END_VAR
VAR_INPUT
	bWlaczPrzyciski								: BOOL;
END_VAR
    Rectangle (0,0 901x401)
    Rectangle (10,10 881x241)
    Frame (210,20 114x44), invisible if: not GVL_StanMaszyny.fbStanMaszyny.arrVisuTryb[GVL_StanMaszyny.fbStanMaszyny.iNumerTrybuPracy][12]
        shows Visu_StanMaszyny_AktualyStan(bNacisniety := GVL_StanMaszyny.fbStanMaszyny.bUnholdingZakonczone, stVisuStan := GVL_StanMaszyny.fbStanMaszyny.arrVisuStany [12])
    Frame (400,20 114x44), invisible if: not GVL_StanMaszyny.fbStanMaszyny.arrVisuTryb[GVL_StanMaszyny.fbStanMaszyny.iNumerTrybuPracy][11]
        shows Visu_StanMaszyny_AktualyStan_BezNaciskania(stVisuStan := GVL_StanMaszyny.fbStanMaszyny.arrVisuStany [11])
    Frame (580,20 114x44), invisible if: not GVL_StanMaszyny.fbStanMaszyny.arrVisuTryb[GVL_StanMaszyny.fbStanMaszyny.iNumerTrybuPracy][10]
        shows Visu_StanMaszyny_AktualyStan(bNacisniety := GVL_StanMaszyny.fbStanMaszyny.bHoldingZakonczone, stVisuStan := GVL_StanMaszyny.fbStanMaszyny.arrVisuStany [10])
    Frame (20,110 114x44), invisible if: not GVL_StanMaszyny.fbStanMaszyny.arrVisuTryb[GVL_StanMaszyny.fbStanMaszyny.iNumerTrybuPracy][4]
        shows Visu_StanMaszyny_AktualyStan_BezNaciskania(stVisuStan := GVL_StanMaszyny.fbStanMaszyny.arrVisuStany [4])
    Frame (210,110 114x44), invisible if: not GVL_StanMaszyny.fbStanMaszyny.arrVisuTryb[GVL_StanMaszyny.fbStanMaszyny.iNumerTrybuPracy][3]
        shows Visu_StanMaszyny_AktualyStan(bNacisniety := GVL_StanMaszyny.fbStanMaszyny.bStartingZakonczone, stVisuStan := GVL_StanMaszyny.fbStanMaszyny.arrVisuStany [3])
    Frame (400,110 114x44), invisible if: not GVL_StanMaszyny.fbStanMaszyny.arrVisuTryb[GVL_StanMaszyny.fbStanMaszyny.iNumerTrybuPracy][6]
        shows Visu_StanMaszyny_AktualyStan_BezNaciskania(stVisuStan := GVL_StanMaszyny.fbStanMaszyny.arrVisuStany [6])
    Frame (580,110 114x44), invisible if: not GVL_StanMaszyny.fbStanMaszyny.arrVisuTryb[GVL_StanMaszyny.fbStanMaszyny.iNumerTrybuPracy][16]
        shows Visu_StanMaszyny_AktualyStan(bNacisniety := GVL_StanMaszyny.fbStanMaszyny.bCompletingZakonczone, stVisuStan := GVL_StanMaszyny.fbStanMaszyny.arrVisuStany [16])
    Frame (765,110 114x44), invisible if: not GVL_StanMaszyny.fbStanMaszyny.arrVisuTryb[GVL_StanMaszyny.fbStanMaszyny.iNumerTrybuPracy][17]
        shows Visu_StanMaszyny_AktualyStan_BezNaciskania(stVisuStan := GVL_StanMaszyny.fbStanMaszyny.arrVisuStany [17])
    Frame (20,200 114x44), invisible if: not GVL_StanMaszyny.fbStanMaszyny.arrVisuTryb[GVL_StanMaszyny.fbStanMaszyny.iNumerTrybuPracy][15]
        shows Visu_StanMaszyny_AktualyStan(bNacisniety := GVL_StanMaszyny.fbStanMaszyny.bResetingSkonczone, stVisuStan := GVL_StanMaszyny.fbStanMaszyny.arrVisuStany [15])
    Frame (210,200 114x44), invisible if: not GVL_StanMaszyny.fbStanMaszyny.arrVisuTryb[GVL_StanMaszyny.fbStanMaszyny.iNumerTrybuPracy][14]
        shows Visu_StanMaszyny_AktualyStan(bNacisniety := GVL_StanMaszyny.fbStanMaszyny.bUnsuspendingZakonczone, stVisuStan := GVL_StanMaszyny.fbStanMaszyny.arrVisuStany [14])
    Frame (400,200 114x44), invisible if: not GVL_StanMaszyny.fbStanMaszyny.arrVisuTryb[GVL_StanMaszyny.fbStanMaszyny.iNumerTrybuPracy][5]
        shows Visu_StanMaszyny_AktualyStan_BezNaciskania(stVisuStan := GVL_StanMaszyny.fbStanMaszyny.arrVisuStany [5])
    Frame (580,200 114x44), invisible if: not GVL_StanMaszyny.fbStanMaszyny.arrVisuTryb[GVL_StanMaszyny.fbStanMaszyny.iNumerTrybuPracy][13]
        shows Visu_StanMaszyny_AktualyStan(bNacisniety := GVL_StanMaszyny.fbStanMaszyny.bSuspendingZakonczone, stVisuStan := GVL_StanMaszyny.fbStanMaszyny.arrVisuStany [13])
    Frame (20,340 114x44), invisible if: not GVL_StanMaszyny.fbStanMaszyny.arrVisuTryb[GVL_StanMaszyny.fbStanMaszyny.iNumerTrybuPracy][2]
        shows Visu_StanMaszyny_AktualyStan_BezNaciskania(stVisuStan := GVL_StanMaszyny.fbStanMaszyny.arrVisuStany [2])
    Frame (210,340 114x44), invisible if: not GVL_StanMaszyny.fbStanMaszyny.arrVisuTryb[GVL_StanMaszyny.fbStanMaszyny.iNumerTrybuPracy][7]
        shows Visu_StanMaszyny_AktualyStan(bNacisniety := GVL_StanMaszyny.fbStanMaszyny.bStoppingZakonczone, stVisuStan := GVL_StanMaszyny.fbStanMaszyny.arrVisuStany [7])
    Frame (400,340 114x44), invisible if: not GVL_StanMaszyny.fbStanMaszyny.arrVisuTryb[GVL_StanMaszyny.fbStanMaszyny.iNumerTrybuPracy][1]
        shows Visu_StanMaszyny_AktualyStan(bNacisniety := GVL_StanMaszyny.fbStanMaszyny.bClearingZakonczone, stVisuStan := GVL_StanMaszyny.fbStanMaszyny.arrVisuStany [1])
    Rectangle (550,320 351x81)
    Frame (580,340 114x44), invisible if: not GVL_StanMaszyny.fbStanMaszyny.arrVisuTryb[GVL_StanMaszyny.fbStanMaszyny.iNumerTrybuPracy][9]
        shows Visu_StanMaszyny_AktualyStan_BezNaciskania(stVisuStan := GVL_StanMaszyny.fbStanMaszyny.arrVisuStany [9])
    Frame (765,340 114x44), invisible if: not GVL_StanMaszyny.fbStanMaszyny.arrVisuTryb[GVL_StanMaszyny.fbStanMaszyny.iNumerTrybuPracy][8]
        shows Visu_StanMaszyny_AktualyStan(bNacisniety := GVL_StanMaszyny.fbStanMaszyny.bAbortingZakonczone, stVisuStan := GVL_StanMaszyny.fbStanMaszyny.arrVisuStany [8])
END_VISUALIZATION

// ---- POUs/90 - Stan Maszyny/Visu/Visu_StanMaszyny_DiagramZPrzyciskami.TcVIS
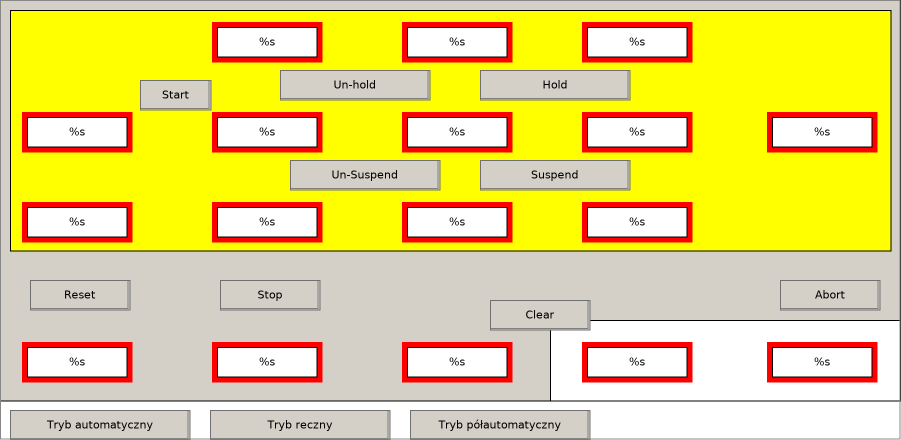
VISUALIZATION Visu_StanMaszyny_DiagramZPrzyciskami  // 901x440
VAR_IN_OUT
	
END_VAR
VAR_INPUT
	bWlaczPrzyciski								: BOOL;
END_VAR
    Frame (0,0 901x401)
        shows Visu_StanMaszyny_Diagram(bWlaczPrzyciski := bWlaczPrzyciski)
    Button (140,80 71x30), "Start", colour toggle: GVL_Elementy.fbPrzysciskStart.bPodswietlenie
        tap GVL_StanMaszyny.bStart
    Button (220,280 100x30), "Stop", colour toggle: GVL_Elementy.fbPrzyciskStop.bPodswietlenie
        tap GVL_StanMaszyny.bStop
    Button (30,280 100x30), "Reset"
        tap GVL_StanMaszyny.bReset
    Button (780,280 100x30), "Abort"
        tap GVL_StanMaszyny.bAbort
    Button (480,70 150x30), "Hold", invisible if: not GVL_StanMaszyny.fbStanMaszyny.arrVisuTryb[GVL_StanMaszyny.fbStanMaszyny.iNumerTrybuPracy][11]
        tap GVL_StanMaszyny.bHold
    Button (280,70 150x30), "Un-hold", invisible if: not GVL_StanMaszyny.fbStanMaszyny.arrVisuTryb[GVL_StanMaszyny.fbStanMaszyny.iNumerTrybuPracy][11]
        tap GVL_StanMaszyny.bUnhold
    Button (480,160 150x30), "Suspend", invisible if: not GVL_StanMaszyny.fbStanMaszyny.arrVisuTryb[GVL_StanMaszyny.fbStanMaszyny.iNumerTrybuPracy][5]
        tap GVL_StanMaszyny.bSuspend
    Button (290,160 150x30), "Un-Suspend", invisible if: not GVL_StanMaszyny.fbStanMaszyny.arrVisuTryb[GVL_StanMaszyny.fbStanMaszyny.iNumerTrybuPracy][5]
        tap GVL_StanMaszyny.bUnsuspend
    Button (10,410 180x30), "Tryb automatyczny", colour toggle: GVL_StanMaszyny.eTrybPracy = E_PMLUnitMode.AUTOMATIC, input disabled if: not (GVL_StanMaszyny.fbStanMaszyny.eStan = E_PMLState.ABORTED or GVL_StanMaszyny.fbStanMaszyny.eStan = E_PMLState.STOPPED)
        OnMouseDown: execute { GVL_StanMaszyny.eTrybPracy	:= E_PMLUnitMode.AUTOMATIC; }
    Button (210,410 180x30), "Tryb reczny", colour toggle: GVL_StanMaszyny.eTrybPracy = E_PMLUnitMode.MANUAL, input disabled if: not (GVL_StanMaszyny.fbStanMaszyny.eStan = E_PMLState.ABORTED or GVL_StanMaszyny.fbStanMaszyny.eStan = E_PMLState.STOPPED)
        OnMouseDown: execute { GVL_StanMaszyny.eTrybPracy	:= E_PMLUnitMode.MANUAL; }
    Button (490,300 100x30), "Clear"
        tap GVL_StanMaszyny.bClear
    Button (410,410 180x30), "Tryb półautomatyczny", colour toggle: GVL_StanMaszyny.eTrybPracy = E_PMLUnitMode.SEMIAUTOMATIC, input disabled if: not (GVL_StanMaszyny.fbStanMaszyny.eStan = E_PMLState.ABORTED or GVL_StanMaszyny.fbStanMaszyny.eStan = E_PMLState.STOPPED)
        OnMouseDown: execute { GVL_StanMaszyny.eTrybPracy	:= E_PMLUnitMode.SEMIAUTOMATIC; }
END_VISUALIZATION

// ---- POUs/95 - Logowanie bledow/Wizualizacja/Visu_LogowanieBledow_Tabela.TcVIS
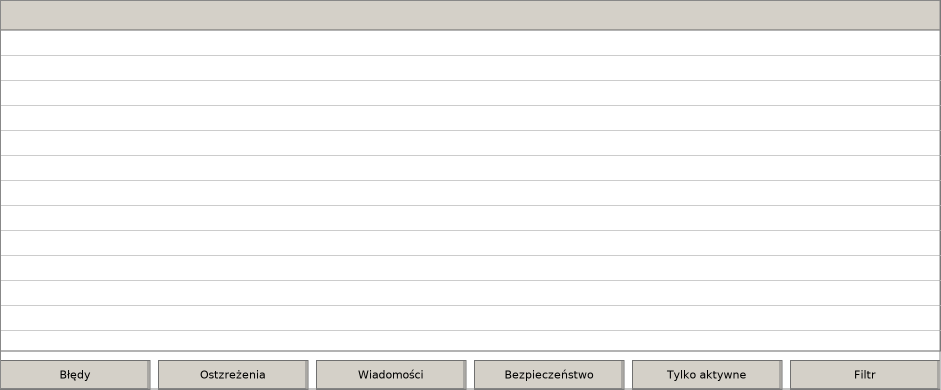
VISUALIZATION Visu_LogowanieBledow_Tabela  // 941x390
VAR_IN_OUT
	stParametry								: DUT_LogowanieBledow_WyswietlanieParametry;
END_VAR
    Table (0,0 941x351), data array: GVL_LogowanieBledow.fbLoger.arrTablicaWyswietlana
        p3854506369: GVL_LogowanieBledow.fbLoger.arrTablicaWyswietlana[INDEX].sNrKomponentu
        p1892666644: GVL_LogowanieBledow.fbLoger.arrTablicaWyswietlana[INDEX].sKodBledu
        p338671338: GVL_LogowanieBledow.fbLoger.arrTablicaWyswietlana[INDEX].byRodzajZdarzenia
        p2170511999: GVL_LogowanieBledow.fbLoger.arrTablicaWyswietlana[INDEX].sOpis
        p3723444502: GVL_LogowanieBledow.fbLoger.arrTablicaWyswietlana[INDEX].dtDataStart
        p1218418051: GVL_LogowanieBledow.fbLoger.arrTablicaWyswietlana[INDEX].dtDataKoniec
        p746581629: GVL_LogowanieBledow.fbLoger.arrTablicaWyswietlana[INDEX].dwKolor
        p2232123230: Nr Elem.
        p2237128397: Data start
        p505689113: Data koniec
        Columns.Column.[3].Template: 16#FF000000 OR (GVL_LogowanieBledow.fbLoger.arrTablicaWyswietlana[INDEX].dwKolor)
    Button (632,360 150x30), "Tylko aktywne", colour toggle: stParametry.bFiltrAktywne
        toggle stParametry.bFiltrAktywne
    Button (0,360 150x30), "Błędy", colour toggle: stParametry.bFiltrRodzaj and stParametry.byFiltrRodzaj = 1
        OnMouseDown: execute {
            (*
            IF (NOT stParametry.bFiltrRodzaj) THEN
            	stParametry.bFiltrRodzaj := TRUE;
            	stParametry.byFiltrRodzaj := 1;
            ELSE
            	stParametry.bFiltrRodzaj := FALSE;
            END_IF
            *)
        }
    Button (158,360 150x30), "Ostzreżenia", colour toggle: stParametry.bFiltrRodzaj and stParametry.byFiltrRodzaj = 2
        OnMouseDown: execute {
            (*
            IF (NOT stParametry.bFiltrRodzaj) THEN
            	stParametry.bFiltrRodzaj := TRUE;
            	stParametry.byFiltrRodzaj := 2;
            ELSE
            	stParametry.bFiltrRodzaj := FALSE;
            END_IF
            *)
        }
    Button (316,360 150x30), "Wiadomości", colour toggle: stParametry.bFiltrRodzaj and stParametry.byFiltrRodzaj = 3
        OnMouseDown: execute {
            (*
            IF (NOT stParametry.bFiltrRodzaj) THEN
            	stParametry.bFiltrRodzaj := TRUE;
            	stParametry.byFiltrRodzaj := 3;
            ELSE
            	stParametry.bFiltrRodzaj := FALSE;
            END_IF
            *)
        }
    Button (474,360 150x30), "Bezpieczeństwo", colour toggle: stParametry.bFiltrRodzaj and stParametry.byFiltrRodzaj = 4
        OnMouseDown: execute {
            (*
            IF (NOT stParametry.bFiltrRodzaj) THEN
            	stParametry.bFiltrRodzaj := TRUE;
            	stParametry.byFiltrRodzaj := 4;
            ELSE
            	stParametry.bFiltrRodzaj := FALSE;
            END_IF
            *)
        }
    Button (790,360 150x30), "Filtr"
END_VISUALIZATION

// ---- VISUs/OknoGlowne.TcVIS
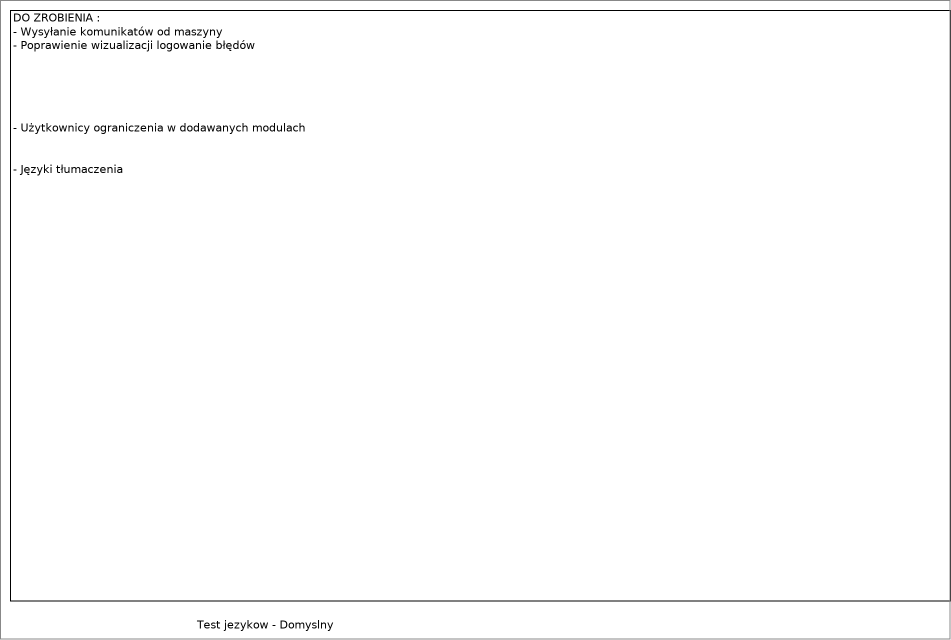
VISUALIZATION OknoGlowne  // 951x640
    Rectangle (10,10 941x591), "DO ZROBIENIA : - Wysyłanie komunikatów od maszyny - Poprawienie wizualizacji logowanie błędów - Użytkownicy ograniczenia w dodawanych modulach - Języki tłumaczenia"
    Label (50,610 431x30), "Test jezykow - Domyslny"
END_VISUALIZATION

// ---- VISUs/Symulacja.TcVIS
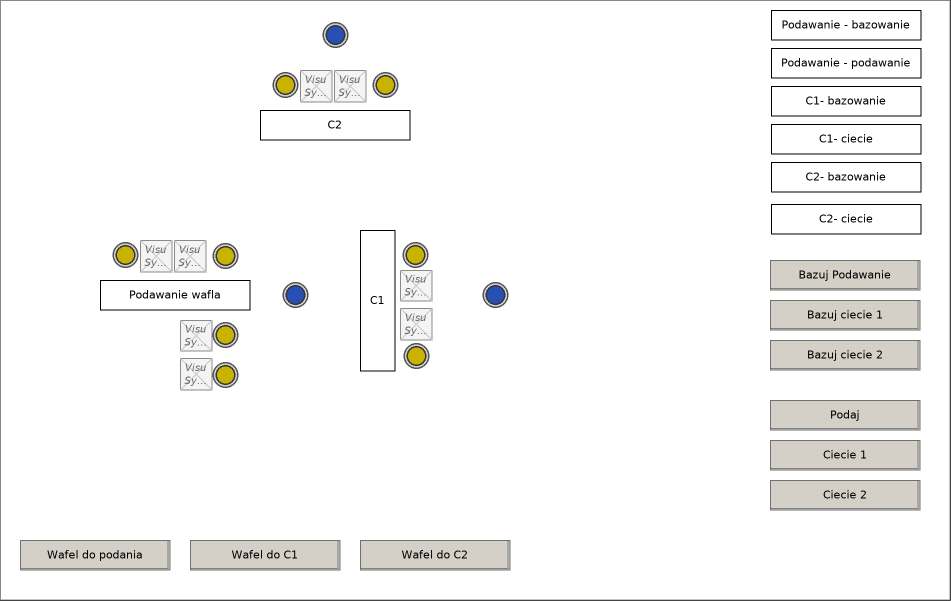
VISUALIZATION Symulacja  // 951x601
VAR_IN_OUT
	stDane									: DUT_Wizualizacja_SymulacjaDane;
END_VAR
    Line (950,0) (950,600)
    Line (0,600) (950,600)
    Rectangle (100,280 150x30), "Podawanie wafla"
    Rectangle (360,230 35x141), "C1"
    Rectangle (260,110 150x30), "C2"
    Lamp1 (401,341 31x30), variable: stDane.bCiecie1_Poczatek, style: Lamp-Lamp1-Yellow
    Lamp1 (400,240 31x30), variable: stDane.bCiecie1_Koniec, style: Lamp-Lamp1-Yellow
    Lamp1 (270,70 31x30), variable: stDane.bCiecie2_Poczatek, style: Lamp-Lamp1-Yellow
    Lamp1 (370,70 31x30), variable: stDane.bCiecie2_Koniec, style: Lamp-Lamp1-Yellow
    Lamp1 (110,240 31x30), variable: stDane.bPodawaniePrzesuwanieKoniec, style: Lamp-Lamp1-Yellow
    Lamp1 (210,241 31x30), variable: stDane.bPodawaniePrzesuwaniePoczatek, style: Lamp-Lamp1-Yellow
    Lamp1 (210,320 31x30), variable: stDane.bPodawanieZabierakKoniec, style: Lamp-Lamp1-Yellow
    Lamp1 (210,360 31x30), variable: stDane.bPodawanieZabierakPoczatek, style: Lamp-Lamp1-Yellow
    Lamp1 (280,280 31x30), variable: stDane.bCzujnikWaflaDoPodania, style: Lamp-Lamp1-Blue
    Lamp1 (480,280 31x30), variable: stDane.bCzujnikWaflaDoCiecia1, style: Lamp-Lamp1-Blue
    Lamp1 (320,20 31x30), variable: stDane.bCzujnikWaflaDoCiecia2, style: Lamp-Lamp1-Blue
    Rectangle (771,10 150x30), "Podawanie - bazowanie", colour toggle: stDane.stStanySilownikow.bPodawanie_Bazowanie
    Rectangle (771,48 150x30), "Podawanie - podawanie", colour toggle: stDane.stStanySilownikow.bPodawanie_Podawanie
    Rectangle (771,86 150x30), "C1- bazowanie", colour toggle: stDane.stStanySilownikow.bCiecie1_Bazowanie
    Rectangle (771,124 150x30), "C1- ciecie", colour toggle: stDane.stStanySilownikow.bCiecie1_Ciecie
    Rectangle (771,162 150x30), "C2- bazowanie", colour toggle: stDane.stStanySilownikow.bCiecie2_Bazowanie
    Rectangle (771,204 150x30), "C2- ciecie", colour toggle: stDane.stStanySilownikow.bCiecie2_Ciecie
    Image (180,358 32x32), invisible if: Not stDane.stStanySilownikow.bPodawanie_Zabierak_WStronePoczatku, image: VisuSymbols.Symbols.ArrowBoldDown
    Image (180,320 32x31), invisible if: Not stDane.stStanySilownikow.bPodawanie_zabierak_WStroneKonca, image: VisuSymbols.Symbols.ArrowBoldUp
    Image (140,240 32x32), invisible if: Not stDane.stStanySilownikow.bPodawanie_Przesuwanie_WStroneKonca, image: VisuSymbols.Symbols.ArrowBoldLeft
    Image (174,240 32x32), invisible if: Not stDane.stStanySilownikow.bPodawanie_Przesuwanie_WStronePoczatku, image: VisuSymbols.Symbols.ArrowBoldRight
    Image (400,308 32x32), invisible if: Not stDane.stStanySilownikow.bCiecie1_Naped_WStronePoczatku, image: VisuSymbols.Symbols.ArrowBoldDown
    Image (400,270 32x31), invisible if: Not stDane.stStanySilownikow.bCiecie1_Naped_WStroneKonca, image: VisuSymbols.Symbols.ArrowBoldUp
    Image (300,70 32x32), invisible if: Not stDane.stStanySilownikow.bCiecie2_Naped_WStronePoczatku, image: VisuSymbols.Symbols.ArrowBoldLeft
    Image (334,70 32x32), invisible if: Not stDane.stStanySilownikow.bCiecie2_Naped_WStroneKonca, image: VisuSymbols.Symbols.ArrowBoldRight
    Button (770,260 150x30), "Bazuj Podawanie", invisible if: stDane.eTrybPracy <> E_PMLUnitMode.SEMIAUTOMATIC
        tap stDane.bPodawanieBazuj
    Button (770,300 150x30), "Bazuj ciecie 1", invisible if: stDane.eTrybPracy <> E_PMLUnitMode.SEMIAUTOMATIC
        tap stDane.bCiecie1Bazuj
    Button (770,340 150x30), "Bazuj ciecie 2", invisible if: stDane.eTrybPracy <> E_PMLUnitMode.SEMIAUTOMATIC
        tap stDane.bCiecie2Bazuj
    Button (770,400 150x30), "Podaj", invisible if: stDane.eTrybPracy <> E_PMLUnitMode.SEMIAUTOMATIC
        tap stDane.bPodawaniePodaj
    Button (770,440 150x30), "Ciecie 1", invisible if: stDane.eTrybPracy <> E_PMLUnitMode.SEMIAUTOMATIC
        tap stDane.bCiecie1Tnij
    Button (770,480 150x30), "Ciecie 2", invisible if: stDane.eTrybPracy <> E_PMLUnitMode.SEMIAUTOMATIC
        tap stDane.bCiecie2Tnij
    Button (20,540 150x30), "Wafel do podania", invisible if: stDane.eTrybPracy <> E_PMLUnitMode.SEMIAUTOMATIC
        toggle stDane.bCzujnikWaflaDoPodania
    Button (190,540 150x30), "Wafel do C1", invisible if: stDane.eTrybPracy <> E_PMLUnitMode.SEMIAUTOMATIC
        toggle stDane.bCzujnikWaflaDoCiecia1
    Button (360,540 150x30), "Wafel do C2", invisible if: stDane.eTrybPracy <> E_PMLUnitMode.SEMIAUTOMATIC
        toggle stDane.bCzujnikWaflaDoCiecia2
END_VISUALIZATION

// ---- VISUs/Ustawienia.TcVIS
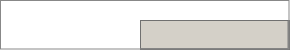
VISUALIZATION Ustawienia  // 290x50
    Button (140,20 150x30)
END_VISUALIZATION

// ---- VISUs/Visualization.TcVIS
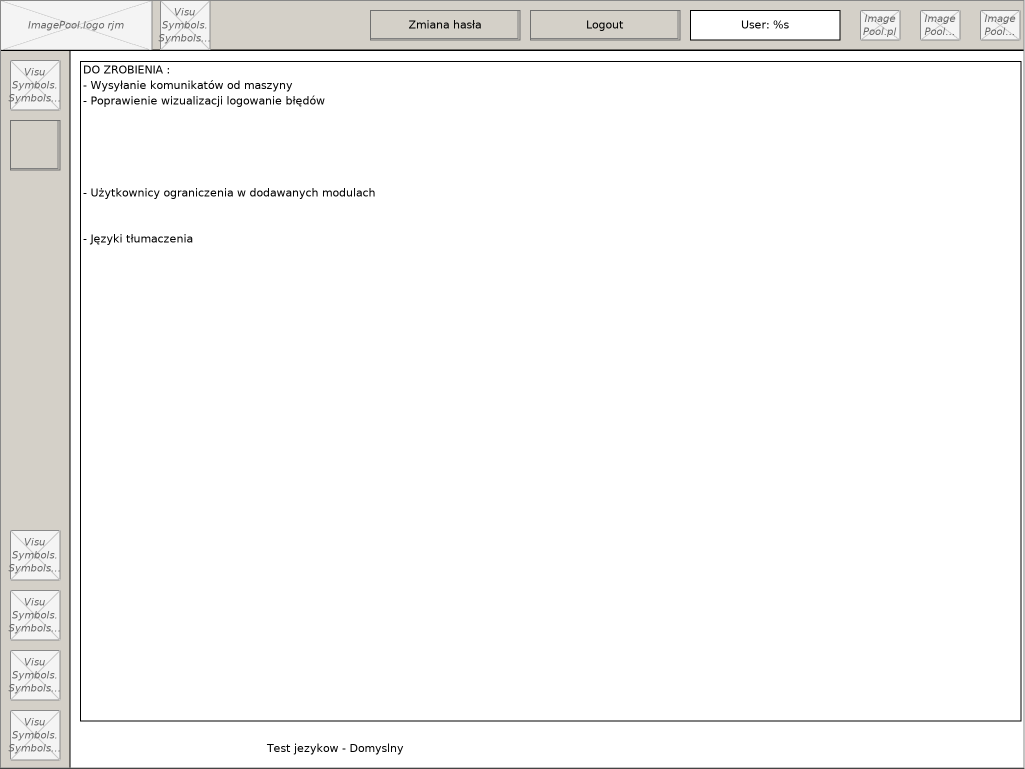
VISUALIZATION Visualization  // 1025x769
    Rectangle (0,0 1024x50)
    Rectangle (0,50 70x718)
    Frame (70,50 951x715), frame switch variable: GVL_Wizualizacja.iNumerRamki
        shows OknoGlowne()
        shows Visu_StanMaszyny_DiagramZPrzyciskami(bWlaczPrzyciski := GVL_StanMaszyny.bWlaczPrzyciski)
        shows Visu_LogowanieBledow_Tabela(stParametry := GVL_LogowanieBledow.fbLoger.stWyswietlanieParametry)
        shows Ustawienia()
        shows Symulacja(stDane := MAIN.fbWizualizacja.stDane)
    Button (10,60 50x50), colour toggle: GVL_Wizualizacja.iNumerRamki = 0
    Button (10,710 50x50), colour toggle: GVL_Wizualizacja.iNumerRamki = 2
    Button (10,650 50x50), colour toggle: GVL_Wizualizacja.iNumerRamki = 1
    Image (10,60 50x50), colour toggle: GVL_Wizualizacja.iNumerRamki = 0, image: VisuSymbols.Symbols.Home
        OnMouseDown: execute {
            GVL_Wizualizacja.iNumerRamki := 0;
            GVL_StanMaszyny.bWlaczPrzyciski := FALSE;
            GVL_LogowanieBledow.bWyswietlAlarmy := FALSE;
        }
    Image (10,650 50x50), image: VisuSymbols.Symbols.Information
        OnMouseDown: execute {
            GVL_Wizualizacja.iNumerRamki := 1;
            GVL_StanMaszyny.bWlaczPrzyciski := TRUE;
            GVL_LogowanieBledow.bWyswietlAlarmy := FALSE;
        }
    Image (10,710 50x50), image: VisuSymbols.Symbols.Security
        OnMouseDown: execute {
            GVL_Wizualizacja.iNumerRamki := 2;
            GVL_StanMaszyny.bWlaczPrzyciski := FALSE;
            GVL_LogowanieBledow.bWyswietlAlarmy := TRUE;
        }
    Image (160,0 50x50), image: VisuSymbols.Symbols.voltage
    Line (0,768) (1024,768)
    Line (1024,768) (1024,0)
    Button (10,590 50x50), colour toggle: GVL_Wizualizacja.iNumerRamki = 3
    Image (10,590 50x50), image: VisuSymbols.Symbols.ControlPanel
        OnMouseDown: execute {
            GVL_Wizualizacja.iNumerRamki := 3;
            GVL_StanMaszyny.bWlaczPrzyciski := FALSE;
            GVL_LogowanieBledow.bWyswietlAlarmy := FALSE;
        }
    Image (0,0 152x50), image: ImagePool.logo rjm
    Line (0,50) (1024,50)
    Image (920,10 40x30), image: ImagePool.de
        OnMouseDown: ChangeLanguage ChangeLanguage=DE
        OnMouseDown: execute { GVL_LogowanieBledow.fbLoger.iJezykID := 1031; }
    Image (980,10 40x30), image: ImagePool.gb
        OnMouseDown: ChangeLanguage ChangeLanguage=EN
        OnMouseDown: execute { GVL_LogowanieBledow.fbLoger.iJezykID := 1033; }
    Image (860,10 40x30), image: ImagePool.pl
        OnMouseDown: execute { GVL_LogowanieBledow.fbLoger.iJezykID := 1045; }
        OnMouseDown: ChangeLanguage ChangeLanguage=PL
    Button (530,10 150x30), "Login", invisible if: VisuElemsWinControls.CurrentUserName <> ""
        OnMouseDown: VisuUserMgmt Type=Login
    Button (530,10 150x30), "Logout", invisible if: VisuElemsWinControls.CurrentUserName = ""
        OnMouseDown: VisuUserMgmt Type=Logout
    Rectangle (690,10 150x30), "User: %s", text variable: VisuElemsWinControls.CurrentUserName
    Button (370,10 150x30), "Zmiana hasła"
        OnMouseDown: VisuUserMgmt Type=ChangeUserPassword
    Button (10,530 50x50)
    Image (10,530 50x50), image: VisuSymbols.Symbols.EditUser
        OnMouseDown: VisuUserMgmt Type=OpenUserConfiguration
    Button (10,120 50x50), colour toggle: GVL_Wizualizacja.iNumerRamki = 4
        OnMouseDown: execute {
            GVL_Wizualizacja.iNumerRamki := 4;
            GVL_StanMaszyny.bWlaczPrzyciski := FALSE;
            GVL_LogowanieBledow.bWyswietlAlarmy := FALSE;
        }
END_VISUALIZATION
